FUNCTION TryConvert_WORD_TO_BOOL : BOOL
VAR_INPUT
	in : WORD;
	out : REFERENCE TO BOOL;
END_VAR

out := WORD_TO_BOOL(in);
TryConvert_WORD_TO_BOOL := TRUE;

END_FUNCTION

(* stored: Version 1.1.0.1, ProductVersion 3.1.4024.12
   POU TryConvert_WORD_TO_BOOL: Id {c0ea2d7a-48b5-4c99-81bb-cf23fcbcec02}, SpecialFunc None *)
